# EPICS autosave request: iocBoot/iocUSBSSR/auto_settings.req
file "USBSSR08_settings.req", P=$(P)
